FUNCTION_BLOCK FunctionsAndFunctionBlocksex03
VAR_INPUT
	number1 		: number;
	number2 		: number;
END_VAR
VAR_OUTPUT
	sum12 			: number;
	counter 		: number;
END_VAR
VAR
END_VAR

END_FUNCTION_BLOCK

(* stored: Version 1.1.0.1
   POU FunctionsAndFunctionBlocksex03: Id {796b8e3a-ac25-44a9-b77b-3e5d1168ed55}, SpecialFunc None *)
